SUBAPPLICATION Einsatzdauerzaehler (* Subapplication Type *)
  (* Standard: 61499-2 *)
  (* Version 1.0, 2024-04-17, Elias *)
  PACKAGE FBs::SlurryTanker::func::Zaehlermenue;
  IMPORT NVS_Keys::Key_Einsatzdauer_Minuten_Store;
  IMPORT NVS_Keys::Key_Einsatzdauer_Stunden_Store;
  IMPORT test::FBs::Baumsetzer::Constants::DefaultPool;
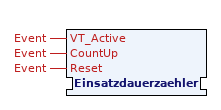
  EVENT_INPUT
    VT_Active;
    CountUp; (* Counts every event *)
    Reset; (* Resets the counter *)
  END_EVENT
  SUBAPPS
    Zaehler_Einsatzdauer : Zaehler_Einsatzdauer(KEY_Std := Key_Einsatzdauer_Stunden_Store, KEY_Min := Key_Einsatzdauer_Minuten_Store, u16ObjId_Std := DefaultPool::NumberVariable_Einsatzdauer_Stunden, u16ObjId_Min := DefaultPool::NumberVariable_Einsatzdauer_Minuten);
  END_SUBAPPS
  EVENT_CONNECTIONS
    CountUp TO Zaehler_Einsatzdauer.CU;
    Reset TO Zaehler_Einsatzdauer.R;
    VT_Active TO Zaehler_Einsatzdauer.rVT;
  END_CONNECTIONS
END_SUBAPPLICATION
